// TIA Portal V20 export
FUNCTION "FC_DBdata" : Void   // FC2, LAD
{ S7_Optimized_Access := 'TRUE' }
// stored: SetENOAutomatically false
   VAR_TEMP
      tempDataReceived : Bool;   // temp flag for 'dataReceived' from FB 'LSql_Microsoft'
      tempAnalyzeDone : Bool;   // temp flag for 'done' from FB 'AnalyzeTokens'
      tempMetaDataAndRowsAvailable : Bool;   // temp flag for 'metaDataAndRowsAvailable' from FB 'AnalyzeTokens'
      queryTemp : String;
   END_VAR
   VAR_TEMP   // added for the SCL form of the ladder/FBD networks
      _w1 : Bool;
   END_VAR
BEGIN

REGION Network 1 (SCL): nel caso la comunicazione con il DB non parte o cadesse, cerco di ripristinarla dopo un timer
   // Check connection to DB and retry to connect if there is a problem

   "DB_executeQuery".timeoutConnection(IN := "SqlConfig".enableLSql AND "SqlConfig".diagnostics.status > 32770 , //8002
                                       PT := T#2s);

   IF "DB_executeQuery".timeoutConnection.Q THEN
       "SqlConfig".enableLSql := false;
   END_IF;

   "DB_executeQuery".timeoutRetrayConnection(IN := NOT "SqlConfig".enableLSql,
                                             PT := T#1s);

   IF "DB_executeQuery".timeoutRetrayConnection.Q THEN
       "SqlConfig".enableLSql := true;
   END_IF;
END_REGION

REGION Network 2: TDS Connection and Communication Handling
   // this network handles the TDS connection and communication
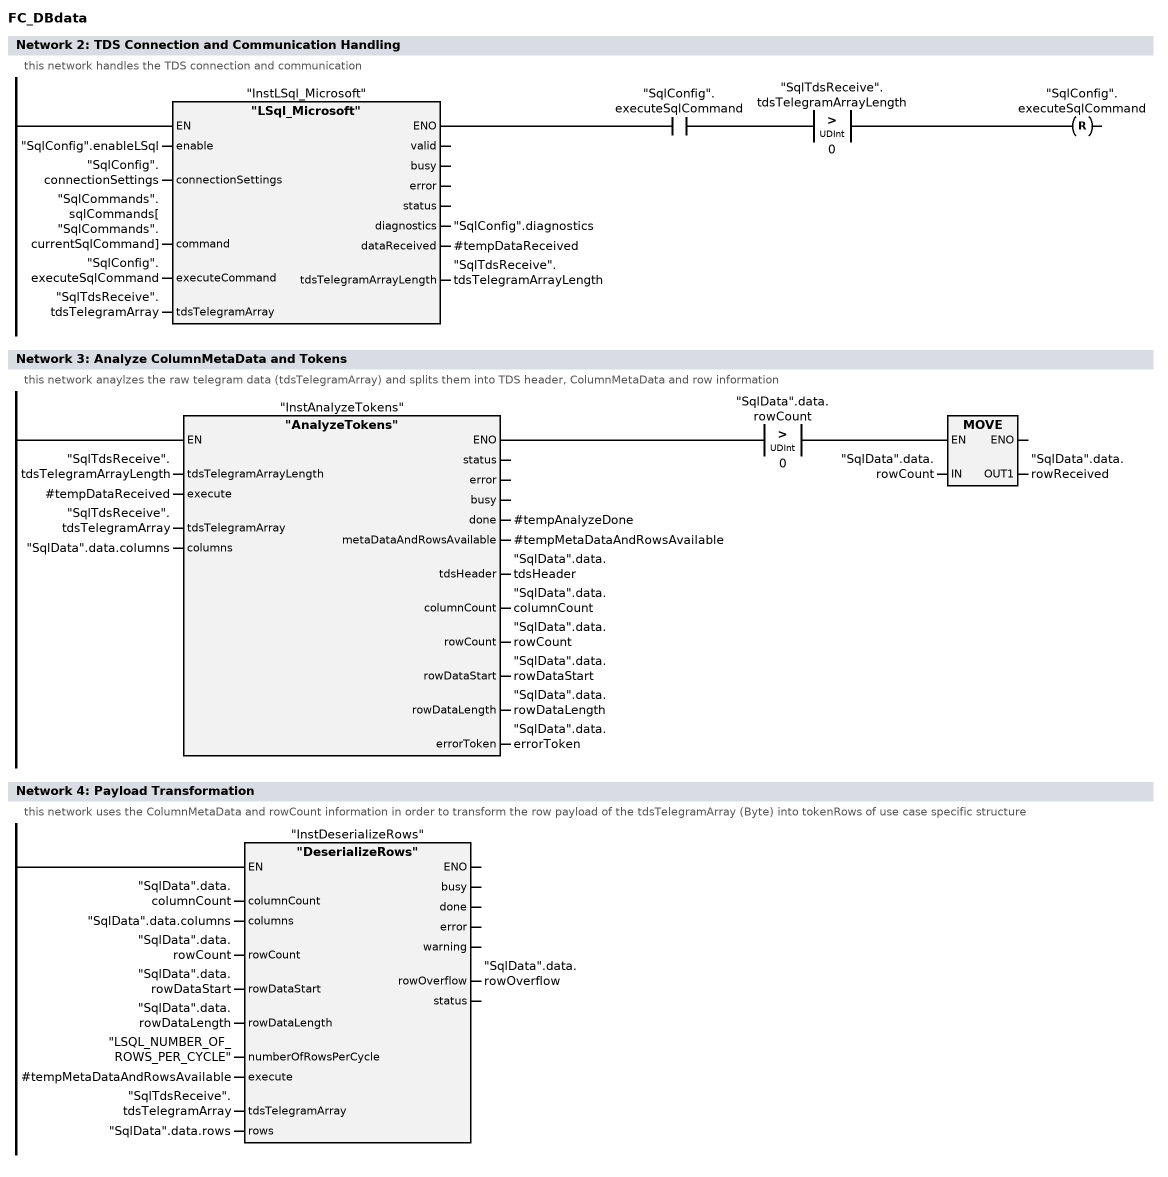
   RUNG wire#powerrail
      "InstLSql_Microsoft"(enable := "SqlConfig".enableLSql, connectionSettings := "SqlConfig".connectionSettings, command := "SqlCommands".sqlCommands["SqlCommands".currentSqlCommand], executeCommand := "SqlConfig".executeSqlCommand, tdsTelegramArray := "SqlTdsReceive".tdsTelegramArray, valid =>, busy =>, error =>, status =>, diagnostics => "SqlConfig".diagnostics, dataReceived => #tempDataReceived, tdsTelegramArrayLength => "SqlTdsReceive".tdsTelegramArrayLength)
      Contact( "SqlConfig".executeSqlCommand )
      { S7_Templates := "SrcType := UDInt" } GT_Contact(in1 := "SqlTdsReceive".tdsTelegramArrayLength, in2 := 0)
      R_Coil( "SqlConfig".executeSqlCommand )
   END_RUNG
   // the same network as SCL:
   "InstLSql_Microsoft"(enable := "SqlConfig".enableLSql,   // "LSql_Microsoft"
                        connectionSettings := "SqlConfig".connectionSettings,
                        command := "SqlCommands".sqlCommands["SqlCommands".currentSqlCommand],
                        executeCommand := "SqlConfig".executeSqlCommand,
                        tdsTelegramArray := "SqlTdsReceive".tdsTelegramArray,
                        diagnostics => "SqlConfig".diagnostics,
                        dataReceived => #tempDataReceived,
                        tdsTelegramArrayLength => "SqlTdsReceive".tdsTelegramArrayLength,
                        ENO => #_w1);
   IF #_w1 AND "SqlConfig".executeSqlCommand AND ("SqlTdsReceive".tdsTelegramArrayLength > 0) THEN
       "SqlConfig".executeSqlCommand := FALSE;
   END_IF;
END_REGION

REGION Network 3: Analyze ColumnMetaData and Tokens
   // this network anaylzes the raw telegram data (tdsTelegramArray) and splits them into TDS header, ColumnMetaData and row information
   RUNG wire#powerrail
      "InstAnalyzeTokens"(tdsTelegramArrayLength := "SqlTdsReceive".tdsTelegramArrayLength, execute := #tempDataReceived, tdsTelegramArray := "SqlTdsReceive".tdsTelegramArray, columns := "SqlData".data.columns, status =>, error =>, busy =>, done => #tempAnalyzeDone, metaDataAndRowsAvailable => #tempMetaDataAndRowsAvailable, tdsHeader => "SqlData".data.tdsHeader, columnCount => "SqlData".data.columnCount, rowCount => "SqlData".data.rowCount, rowDataStart => "SqlData".data.rowDataStart, rowDataLength => "SqlData".data.rowDataLength, errorToken => "SqlData".data.errorToken)
      { S7_Templates := "SrcType := UDInt" } GT_Contact(in1 := "SqlData".data.rowCount, in2 := 0)
      Move(in := "SqlData".data.rowCount, out1 => "SqlData".data.rowReceived)
   END_RUNG
   // the same network as SCL:
   "InstAnalyzeTokens"(tdsTelegramArrayLength := "SqlTdsReceive".tdsTelegramArrayLength,   // "AnalyzeTokens"
                       execute := #tempDataReceived,
                       tdsTelegramArray := "SqlTdsReceive".tdsTelegramArray,
                       columns := "SqlData".data.columns,
                       done => #tempAnalyzeDone,
                       metaDataAndRowsAvailable => #tempMetaDataAndRowsAvailable,
                       tdsHeader => "SqlData".data.tdsHeader,
                       columnCount => "SqlData".data.columnCount,
                       rowCount => "SqlData".data.rowCount,
                       rowDataStart => "SqlData".data.rowDataStart,
                       rowDataLength => "SqlData".data.rowDataLength,
                       errorToken => "SqlData".data.errorToken,
                       ENO => #_w1);
   IF #_w1 AND ("SqlData".data.rowCount > 0) THEN
       "SqlData".data.rowReceived := "SqlData".data.rowCount;
   END_IF;
END_REGION

REGION Network 4: Payload Transformation
   // this network uses the ColumnMetaData and rowCount information in order to transform the row payload of the tdsTelegramArray (Byte) into tokenRows of use case specific structure
   RUNG wire#powerrail
      "InstDeserializeRows"(columnCount := "SqlData".data.columnCount, columns := "SqlData".data.columns, rowCount := "SqlData".data.rowCount, rowDataStart := "SqlData".data.rowDataStart, rowDataLength := "SqlData".data.rowDataLength, numberOfRowsPerCycle := "LSQL_NUMBER_OF_ROWS_PER_CYCLE", execute := #tempMetaDataAndRowsAvailable, tdsTelegramArray := "SqlTdsReceive".tdsTelegramArray, rows := "SqlData".data.rows, busy =>, done =>, error =>, warning =>, rowOverflow => "SqlData".data.rowOverflow, status =>)
   END_RUNG
   // the same network as SCL:
   "InstDeserializeRows"(columnCount := "SqlData".data.columnCount,   // "DeserializeRows"
                         columns := "SqlData".data.columns,
                         rowCount := "SqlData".data.rowCount,
                         rowDataStart := "SqlData".data.rowDataStart,
                         rowDataLength := "SqlData".data.rowDataLength,
                         numberOfRowsPerCycle := "LSQL_NUMBER_OF_ROWS_PER_CYCLE",
                         execute := #tempMetaDataAndRowsAvailable,
                         tdsTelegramArray := "SqlTdsReceive".tdsTelegramArray,
                         rows := "SqlData".data.rows,
                         rowOverflow => "SqlData".data.rowOverflow);
END_REGION
END_FUNCTION
